{attribute 'qualified_only'}
{attribute 'strict'}
TYPE E_TCP_DEVICE_TYPE :
(
	LAKESHORE_224 := 0,
	LAKESHORE_336
);
END_TYPE

(* stored: Version 1.1.0.1, ProductVersion 3.1.4022.16
   DUT E_TCP_DEVICE_TYPE: Id {3757cbf1-3e2a-4682-8f70-146a6ebaffd7} *)
